// TIA Portal V16 export
// export: Created 2021-08-30T13:41:02.0125126Z, ExportSetting WithDefaults, DisplayName Totally Integrated Automation Portal, DisplayVersion V16 Update 3, DisplayName TIA Portal Version Control Interface, DisplayVersion V16 Update 2, DisplayName TIA Portal Openness, DisplayVersion V16 Update 3, DisplayName TIA Portal Teamcenter Gateway, DisplayVersion V16, DisplayName STEP 7 Professional, DisplayVersion V16 Update 3, DisplayName STEP 7 Safety, DisplayVersion V16, DisplayName WinCC Advanced, DisplayVersion V16 Update 3
DATA_BLOCK "AllDpump_DB"   // DB15
VERSION : 0.1
// stored: AutoNumber true, DBAccessibleFromOPCUA true, InstanceOfName AllDpump, InstanceOfType FB
"AllDpump"
   // VAR
   //    dp101 { S7_SetPoint := 'True'} : "DPumpCntr";
   //    dp501 { S7_SetPoint := 'True'} : "DPumpCntr";
   //    dp502 { S7_SetPoint := 'True'} : "DPumpCntr";
   //    dp801 { S7_SetPoint := 'True'} : "DPumpCntr";
   //    dp802 { S7_SetPoint := 'True'} : "DPumpCntr";
   //    dp803 { S7_SetPoint := 'True'} : "DPumpCntr";
   //    dp1001 { S7_SetPoint := 'True'} : "DPumpCntr";
   // END_VAR
BEGIN
END_DATA_BLOCK
